FUNCTION_BLOCK ABSTRACT MockEventHandler IMPLEMENTS I_EventHandler
VAR
	_eventReceived : BOOL;
	fromExpected : BOOL;
END_VAR

PROPERTY PUBLIC EventReceived : BOOL
GET // PUBLIC
EventReceived := _eventReceived;
END_GET
END_PROPERTY

PROPERTY PUBLIC FromExpectedOriginator : BOOL
GET // PUBLIC
FromExpectedOriginator := fromExpected;
END_GET
END_PROPERTY

METHOD PUBLIC ABSTRACT HandleEvent
VAR_INPUT
	Event : mobject_events.I_Event;
END_VAR
END_METHOD

METHOD PUBLIC Reset
_eventReceived := FALSE;
fromExpected := FALSE;
END_METHOD

END_FUNCTION_BLOCK

(* stored: Version 1.1.0.1, ProductVersion 3.1.4024.12
   POU MockEventHandler: Id {1f5b9b53-3872-4edc-a8c7-4143aceb98f1}, SpecialFunc None
   Property EventReceived: Id {63567c50-4334-49ad-b7d0-444b2d50aa57}
   Get Get: Id {2278bf52-901e-454b-8702-86a4ce3b3220}
   Property FromExpectedOriginator: Id {2e61ab88-541e-40bd-85f2-bca1a4a463c6}
   Get Get: Id {feb811a2-267d-4bdf-aa1b-94c0227904ac}
   Method HandleEvent: Id {af9fef76-1c12-41b2-abaa-5e8b57712e00}
   Method Reset: Id {7fe12c68-eab0-4bf3-a3c3-83a0103f11d2} *)
